// TwinCAT 3 PLC project Untitled1
// ProgramVersion: 3.1.4024.0
// libraries:
//   Tc2_MC2, * (Beckhoff Automation GmbH)
//   Tc2_Standard, * (Beckhoff Automation GmbH)
//   Tc2_System, * (Beckhoff Automation GmbH)
//   Tc3_Module, * (Beckhoff Automation GmbH)
//   VisuDialogs, * (System)
//   VisuSymbols,3.5.10.0,System
// project tree:
//   / GlobalTextList.TcGTLO, PlcTask.TcTTO (not stored), Visualization Manager.TcVMO (not stored)
//   GVLs/ BinSensorsFromPlc2.TcGVL, GVL.TcGVL (not stored), Inputs.TcGVL, MeasuringData.TcGVL, OpcuaData.TcGVL, Outputs.TcGVL, Steps.TcGVL
//   POUs/ AxisControl.TcPOU, BreedCalculation.TcPOU, Control24V.TcPOU, MAIN.TcPOU, PLC2Communicaton.TcPOU, SaveNewBinPosition.TcPOU, ServoManualMotion.TcPOU, SizeMeasure.TcPOU, TablePositions.TcPOU, WeightMeasure.TcPOU
//   VISUs/ HMI.TcVIS, InputsScreen.TcVIS, MainScreen.TcVIS, ManualMotionScreen.TcVIS, ServoMotionScreen.TcVIS
// real-time tasks:
//   TASK PlcTask: cycle T#10ms, priority 20, ADS port 350
// motion (NC):
//   TASK NC-Task 1 SAF: cycle T#2ms, priority 4, ADS port 501
//   TASK NC-Task 1 SVB: cycle T#10ms, priority 8, ADS port 511
//   AXIS Axis 1 (id 1)
//     Dynamic: Acceleration=120, Deceleration=120, Jerk=1000
//     Velo: SlowManual=20, FastManual=70, Maximum=150
//     OtherSettings: AllowMotionCmdToSlave=true
//     encoder EncType=1
//       EncPara: ScaleFactorNumerator=1
//         SoftEndMinControl: Enable=true, Range=-500
//         SoftEndMaxControl: Enable=true, Range=500
//     drive DrvType=5
//       Analog: VeloReferenz=100, TorqueSetpointScale=10, ScaleFactorActTorque=0.1
//       TimeComp: TaskDelayCycles=1
//     controller CtrType=1
//       CtrPara: PriorControlFactor=1
//         Observer: BandWidth=20
// variable links:
//   Untitled1/Untitled1 Instance <-> NC-Task 1 SAF/Axes/Axis 1
//     PlcTask Inputs/GVL.Axis.NcToPlc <-> Outputs/ToPlc
//     PlcTask Outputs/GVL.Axis.PlcToNc <-> Inputs/FromPlc

// ---- GVLs/BinSensorsFromPlc2.TcGVL
{attribute 'qualified_only'}
VAR_GLOBAL
	Bin1Full : BOOL := TRUE;
	Bin2Full : BOOL := TRUE;
	Bin3Full : BOOL := TRUE;
	Bin4Full : BOOL := TRUE;

END_VAR

// ---- GVLs/Inputs.TcGVL
{attribute 'qualified_only'}
VAR_GLOBAL
	Start_pos : BOOL;
	Size_measure_pos : BOOL;
	Weight_mes_pos : BOOL;
	Servo_table_pos : BOOL;
	Metal_sensor : BOOL;
	Grip_cyl_end_ext : BOOL;
	Grip_cyl_end_ret : BOOL;
	Cyl_at_table_ext : BOOL;
	Cyl_at_table_ret : BOOL;
	ES1 : BOOL;
	ES2 : BOOL;
	Size_measure : INT;
	Load_cell : INT;
	Grip_cyl_start_ext : BOOL;
	Grip_cyl_start_ret : BOOL;
	Control24VButton : BOOL;
	Metal_measure_pos : BOOL;
	End_pos_at_conveyor : BOOL;
	Item_left_the_table : BOOL;
END_VAR

// ---- GVLs/MeasuringData.TcGVL
{attribute 'qualified_only'}
VAR_GLOBAL
	AutomaticMode : BOOL;		
	StartConveyor : BOOL;	
	StopConveyor : BOOL;		
	ItemInTheSystem : BOOL; //If there is an item in the system
	ItemInTheSystemOnHmi : BOOL := TRUE; //If the variable true the text is invisible
	TableAtHome : BOOL;		
	TableAtBin1 : BOOL;		
	TableAtBin2 : BOOL;		
	TableAtBin3 : BOOL;		
	TableAtBin4 : BOOL;		
	ES1NC : BOOL := TRUE; //Emergency button for simulation
	ES2NC : BOOL := TRUE; //Emergency button for simulation
	ControlSupplyOK : BOOL; //Control 24V for simulation
	ControlSupplyOKOnHmi : BOOL := TRUE; //If the variable true the text is invisible
	SizeInCm : REAL;		
	MetalMaterial : BOOL;		
	WeightInKg : REAL;	
	Bin1Breed : BOOL; //Small and non metal
	Bin2Breed : BOOL; //Small and metal
	Bin3Breed : BOOL; //Large and not metal
	Bin4Breed : BOOL; //Large and metal
	Bin1BreedOnHmi : BOOL := TRUE; //If the variable true the text is invisible
	Bin2BreedOnHmi : BOOL := TRUE; //If the variable true the text is invisible
	Bin3BreedOnHmi : BOOL := TRUE; //If the variable true the text is invisible
	Bin4BreedOnHmi : BOOL := TRUE; //If the variable true the text is invisible
	HomePosition : LREAL;	
	Bin1Position : LREAL := 30.0;		
	Bin2Position : LREAL := 60.0;		
	Bin3Position : LREAL := 90.0;		
	Bin4Position : LREAL := 120.0;	
	MoveToBin1PositionByManual : BOOL;		
	MoveToBin2PositionByManual : BOOL;		
	MoveToBin3PositionByManual : BOOL;		
	MoveToBin4PositionByManual : BOOL;		
	MoveToHomeByManual : BOOL;		
	SaveNewPositionOfBin1 : BOOL;	
	SaveNewPositionOfBin2 : BOOL;		
	SaveNewPositionOfBin3 : BOOL;		
	SaveNewPositionOfBin4 : BOOL;		

END_VAR

// ---- GVLs/OpcuaData.TcGVL
{attribute 'qualified_only'}
VAR_GLOBAL
END_VAR

// ---- GVLs/Outputs.TcGVL
{attribute 'qualified_only'}
VAR_GLOBAL
	Green_light : BOOL;
	Yellow_light : BOOL;
	Red_light : BOOL;
	Move_grip_cyl_end_fwd : BOOL;
	Move_grip_cyl_end_bwd : BOOL;
	Move_cyl_at_table_fwd : BOOL;
	Move_cyl_at_table_bwd : BOOL;
	Conveyor_forward : BOOL;
	Conveyor_backward : BOOL;
	Move_grip_cyl_start_fwd : BOOL;
	Move_grip_cyl_start_bwd : BOOL;
	Blue_light : BOOL;

END_VAR

// ---- GVLs/Steps.TcGVL
{attribute 'qualified_only'}
VAR_GLOBAL
	ActualStep : BYTE := 1;
END_VAR

// ---- POUs/AxisControl.TcPOU
FUNCTION_BLOCK AxisControl
VAR_INPUT
	//Enable
	McPowerEnable : BOOL;
	//Jog
	JogForward : BOOL;
	JogBackward : BOOL;
	JogVelocity : LREAL;
	//Absolute move
	AbsolutePosition : LREAL;
	ExecuteMoveAbsoluteByManual : BOOL;
	ExecuteMoveAbsoluteByAutomatic : BOOL;
	MoveToBin1 : BOOL;
	MoveToBin2 : BOOL;
	MoveToBin3 : BOOL;
	MoveToBin4 : BOOL;
	//Home move
	ExecuteHomeByManual : BOOL;
	ExecuteHomeByAutomatic : BOOL;
END_VAR
VAR_OUTPUT
	//Position
	ActualPosition : LREAL;
	//Velocity
	ActualVelocity : LREAL;
END_VAR
VAR
	//Power
	McPower : MC_Power;
	McPowerError : BOOL;
	AxisStatus : BOOL;
	//JOG
	McJog : MC_Jog;

	//Relative
	McMoveRelative : MC_MoveRelative;
	ExecuteRelative : BOOL;
	RelativeDistance : LREAL;
	RelativeVelocity : LREAL;
	//Absolute
	McMoveAbsolute : MC_MoveAbsolute;
	ExecuteAbsolute : BOOL;
	AbsoluteVelocity : LREAL;
	//Velocity
	McMoveVelocity : MC_MoveVelocity;
	ExecuteVelocity : BOOL;
	Velocity : LREAL;
	//Home
	McHome: MC_Home;
	ExecuteHome : BOOL;
	HomeSensor : BOOL;
	//Stop
	McStop : MC_Stop;
	ExecuteStop : BOOL;
	//Halt
	McHalt: MC_Halt;
	ExecuteHalt : BOOL;
END_VAR

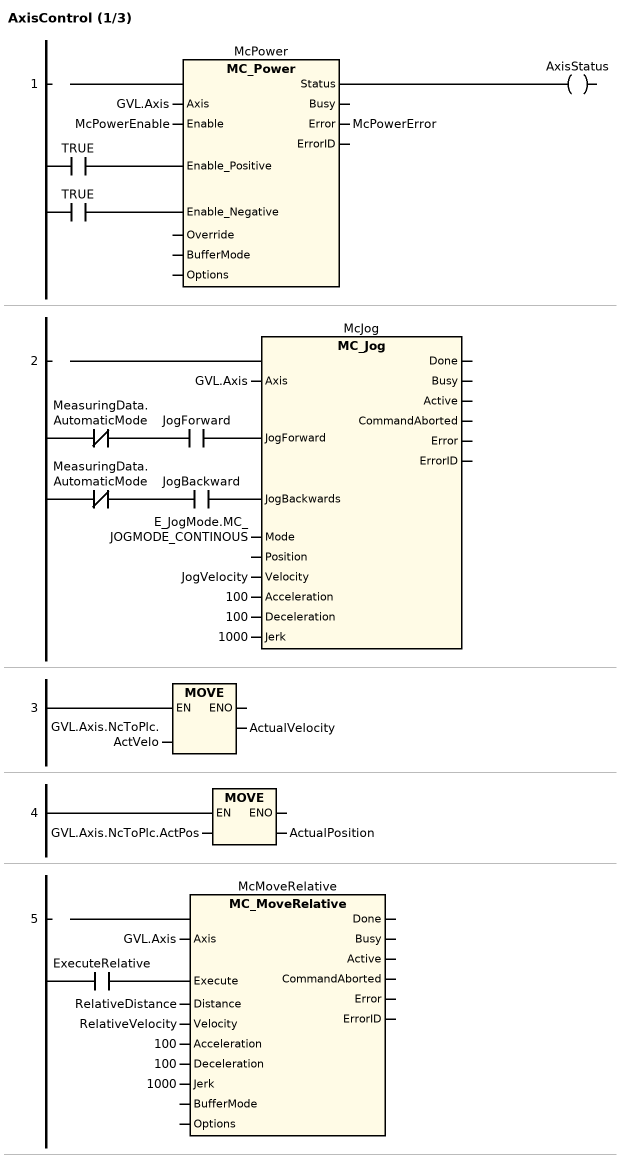
// NETWORK 1
McPower(
    Axis := GVL.Axis,
    Enable := McPowerEnable,
    Enable_Positive := TRUE,
    Enable_Negative := TRUE,
    Error => McPowerError); // MC_Power
AxisStatus := McPower.Status;

// NETWORK 2
McJog(
    Axis := GVL.Axis,
    JogForward := NOT MeasuringData.AutomaticMode AND JogForward,
    JogBackwards := NOT MeasuringData.AutomaticMode AND JogBackward,
    Mode := E_JogMode.MC_JOGMODE_CONTINOUS,
    Velocity := JogVelocity,
    Acceleration := 100,
    Deceleration := 100,
    Jerk := 1000); // MC_Jog

// NETWORK 3
ActualVelocity := GVL.Axis.NcToPlc.ActVelo;

// NETWORK 4
ActualPosition := GVL.Axis.NcToPlc.ActPos;

// NETWORK 5
McMoveRelative(
    Axis := GVL.Axis,
    Execute := ExecuteRelative,
    Distance := RelativeDistance,
    Velocity := RelativeVelocity,
    Acceleration := 100,
    Deceleration := 100,
    Jerk := 1000); // MC_MoveRelative

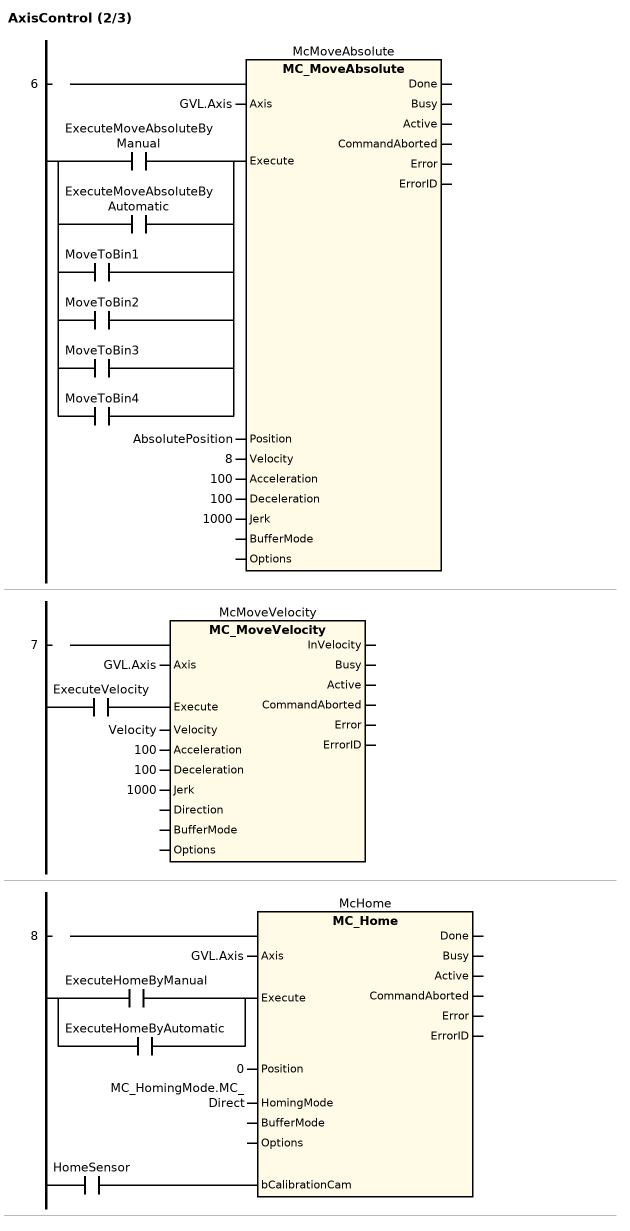
// NETWORK 6
McMoveAbsolute(
    Axis := GVL.Axis,
    Execute := ExecuteMoveAbsoluteByManual OR ExecuteMoveAbsoluteByAutomatic OR MoveToBin1 OR MoveToBin2 OR MoveToBin3 OR MoveToBin4,
    Position := AbsolutePosition,
    Velocity := 8,
    Acceleration := 100,
    Deceleration := 100,
    Jerk := 1000); // MC_MoveAbsolute

// NETWORK 7
McMoveVelocity(
    Axis := GVL.Axis,
    Execute := ExecuteVelocity,
    Velocity := Velocity,
    Acceleration := 100,
    Deceleration := 100,
    Jerk := 1000); // MC_MoveVelocity

// NETWORK 8
McHome(
    Axis := GVL.Axis,
    Execute := ExecuteHomeByManual OR ExecuteHomeByAutomatic,
    Position := 0,
    HomingMode := MC_HomingMode.MC_Direct,
    bCalibrationCam := HomeSensor); // MC_Home

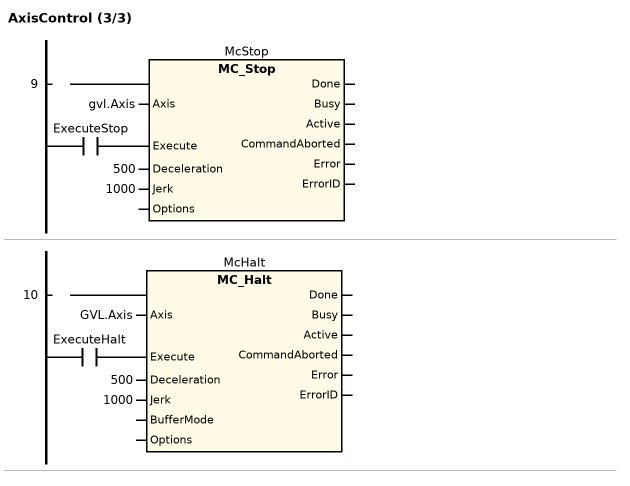
// NETWORK 9
McStop(Axis := gvl.Axis, Execute := ExecuteStop, Deceleration := 500, Jerk := 1000); // MC_Stop

// NETWORK 10
McHalt(Axis := GVL.Axis, Execute := ExecuteHalt, Deceleration := 500, Jerk := 1000); // MC_Halt

END_FUNCTION_BLOCK

// ---- POUs/BreedCalculation.TcPOU
FUNCTION BreedCalculation
VAR_INPUT
END_VAR
VAR

END_VAR


//Small and non metal. Bin1 breed
IF (MAIN.sizeMeasure.sizeInCm >= 10.0 AND MAIN.sizeMeasure.sizeInCm <= 20.0 AND MAIN.weightMeasure.weightInKg <= 5.0 AND
	NOT MeasuringData.MetalMaterial) THEN
	MeasuringData.Bin1Breed := TRUE;
	MeasuringData.Bin2Breed := FALSE;
	MeasuringData.Bin3Breed := FALSE;
	MeasuringData.Bin4Breed := FALSE;
	//Variables on the HMI
	MeasuringData.Bin1BreedOnHmi := FALSE;
	MeasuringData.Bin2BreedOnHmi := TRUE;
	MeasuringData.Bin3BreedOnHmi := TRUE;
	MeasuringData.Bin4BreedOnHmi := TRUE;
END_IF

//Small and metal. Bin2 breed
IF (MAIN.sizeMeasure.sizeInCm >= 10.0 AND MAIN.sizeMeasure.sizeInCm <= 20.0 AND MAIN.weightMeasure.weightInKg <= 5.0 AND
	MeasuringData.MetalMaterial) THEN
	MeasuringData.Bin1Breed := FALSE;
	MeasuringData.Bin2Breed := TRUE;
	MeasuringData.Bin3Breed := FALSE;
	MeasuringData.Bin4Breed := FALSE;
	//Variables on the HMI
	MeasuringData.Bin1BreedOnHmi := TRUE;
	MeasuringData.Bin2BreedOnHmi := FALSE;
	MeasuringData.Bin3BreedOnHmi := TRUE;
	MeasuringData.Bin4BreedOnHmi := TRUE;
END_IF

//Large and non metal. Bin3 breed
IF (MAIN.sizeMeasure.sizeInCm >= 20.0 AND MAIN.weightMeasure.weightInKg >= 5.1 AND
	NOT MeasuringData.MetalMaterial) THEN
	MeasuringData.Bin1Breed := FALSE;
	MeasuringData.Bin2Breed := FALSE;
	MeasuringData.Bin3Breed := TRUE;
	MeasuringData.Bin4Breed := FALSE;
	//Variables on the HMI
	MeasuringData.Bin1BreedOnHmi := TRUE;
	MeasuringData.Bin2BreedOnHmi := TRUE;
	MeasuringData.Bin3BreedOnHmi := FALSE;
	MeasuringData.Bin4BreedOnHmi := TRUE;
END_IF

//Large and metal. Bin4 breed
IF (MAIN.sizeMeasure.sizeInCm >= 20.0 AND MAIN.weightMeasure.weightInKg >= 5.1 AND
	MeasuringData.MetalMaterial) THEN
	MeasuringData.Bin1Breed := FALSE;
	MeasuringData.Bin2Breed := FALSE;
	MeasuringData.Bin3Breed := FALSE;
	MeasuringData.Bin4Breed := TRUE;
	//Variables on the HMI
	MeasuringData.Bin1BreedOnHmi := TRUE;
	MeasuringData.Bin2BreedOnHmi := TRUE;
	MeasuringData.Bin3BreedOnHmi := TRUE;
	MeasuringData.Bin4BreedOnHmi := FALSE;
END_IF

END_FUNCTION

// ---- POUs/MAIN.TcPOU
PROGRAM MAIN
VAR
	AxisControl : AxisControl;
	sizeMeasure : sizeMeasure;
	weightMeasure : WeightMeasure;
	control24V : Control24V;
	
	//Timers
	fbTon1 : TON;
	fbTon2 : TON;
	fbTon3 :TON;
	fbTon4 :TON;
	fbTon5 : TON;
	fbTon6 : TON;
	fbTon7 : TON;
	fbTp1 : TP;
	
	//Falling and rising edges
	startPosFallingEdge : F_TRIG;
	itemLeftTheTableFallingEdge : F_TRIG;
	
END_VAR

AxisControl();
sizeMeasure();
weightMeasure();

//Control 24V power supply
control24V();

//If there is 24V control supply, the servo is ready to operate
IF MeasuringData.ControlSupplyOK THEN
	AxisControl(McPowerEnable := TRUE);
ELSE
	AxisControl(McPowerEnable := FALSE);
END_IF

//Table positions
TablePositions();

//Save new bin position
SaveNewBinPosition();

//Breed calculation
BreedCalculation();

//Manual motion of servo
ServoManualMotion();

//PLC2 communication

//The blue light is on if there is 24V control supply.
IF MeasuringData.ControlSupplyOK THEN
	Outputs.Blue_light := TRUE;
ELSE
	Outputs.Blue_light := FALSE;
END_IF

//Start the system and the conveyor from HMI button.
//The yellow light is on.
IF MeasuringData.AutomaticMode AND MeasuringData.StartConveyor THEN
	fbTon1(IN := TRUE, PT := T#3S);
ELSE
	fbTon1(IN := FALSE);
END_IF

IF fbTon1.Q THEN
	Outputs.Yellow_light := TRUE;
	Outputs.Conveyor_forward := TRUE;
END_IF

//Halt the conveyor
IF MeasuringData.AutomaticMode AND MeasuringData.StopConveyor THEN
	Outputs.Conveyor_forward := FALSE;
END_IF

//Halt the servo motor

//Move gripping cylinder in start position backward.
//If there is no item in the system.
IF Steps.ActualStep = 1 AND Inputs.Start_pos THEN
	fbTon2(IN := TRUE, PT := T#3S);
ELSE
	fbTon2(IN := FALSE);
END_IF

IF fbTon2.Q AND NOT MeasuringData.ItemInTheSystem THEN
	Outputs.Move_grip_cyl_start_bwd := TRUE;
	Steps.ActualStep := 2;
END_IF

//After leaving the start position sensor, the system is in progress so there is an item in the system.
//The green light is on.
//The yellow light is off.
//Move gripping cylinder in start position forward.
startPosFallingEdge(CLK := Inputs.Start_pos);
IF startPosFallingEdge.Q THEN
	MeasuringData.ItemInTheSystem := TRUE;
	MeasuringData.ItemInTheSystemOnHmi := FALSE;
	Outputs.Green_light := TRUE;
	Outputs.Yellow_light := FALSE;
	Outputs.Move_grip_cyl_start_bwd := FALSE;
END_IF

//If the sensor active for two seconds, save the size in the data block.
IF Steps.ActualStep = 2 AND Inputs.Size_measure_pos THEN
	fbTon3(IN := TRUE, PT := T#3S);
ELSE
	fbTon3(IN := FALSE);
END_IF

IF fbTon3.Q THEN
	MeasuringData.SizeInCm := sizeMeasure.sizeInCm;
	Steps.ActualStep := 3;
END_IF

//Metal measure
IF Steps.ActualStep = 3 AND Inputs.Metal_measure_pos AND Inputs.Metal_sensor THEN
	MeasuringData.MetalMaterial := TRUE;
	Steps.ActualStep :=4 ;
END_IF

//Weight measure
IF Steps.ActualStep = 4 AND Inputs.Weight_mes_pos THEN
	fbTon4(IN := TRUE, PT := T#2S);
ELSE
	fbTon4(IN := FALSE);
END_IF

IF fbTon4.Q THEN
	MeasuringData.WeightInKg := weightMeasure.weightInKg;
	Steps.ActualStep := 5;
END_IF

//TCP/IP communication between the PLCs.
//If the end position sensor or sensor at the table are active, getting bin saturation data from PLC2.


//Retract gripping cylinder in end position
//If the sensor at conveyor is active for 1.5 seconds and the reed sensor is active and the certain bin is not full and the table is at home position.
//The state of bin sensors comes from PLC2.
IF Steps.ActualStep = 5 AND Inputs.End_pos_at_conveyor THEN
	fbTon5(IN := TRUE, PT := T#1.5S);
ELSE
	fbTon5(IN := FALSE);
END_IF

IF fbTon5.Q AND Inputs.Grip_cyl_end_ext AND MeasuringData.TableAtHome AND
	(
	(MeasuringData.Bin1Breed AND NOT BinSensorsFromPlc2.Bin1Full) OR
	(MeasuringData.Bin2Breed AND NOT BinSensorsFromPlc2.Bin2Full) OR
	(MeasuringData.Bin3Breed AND NOT BinSensorsFromPlc2.Bin3Full) OR
	(MeasuringData.Bin4Breed AND NOT BinSensorsFromPlc2.Bin4Full)
	)
	THEN
	
	Outputs.Move_grip_cyl_end_bwd := TRUE;
	Steps.ActualStep := 6;
END_IF

//Moving the servo controlled table to the appropriate position.
//If the item is already on the table, extending the cylinder in end position.
IF Inputs.Servo_table_pos THEN
	fbTon6(IN := TRUE, PT := T#2S);
ELSE
	fbTon6(IN := FALSE);
END_IF

IF fbTon6.Q THEN
	Outputs.Move_grip_cyl_end_bwd := FALSE;
END_IF

//Move to bin1
IF fbTon6.Q AND MeasuringData.Bin1Breed AND NOT BinSensorsFromPlc2.Bin1Full THEN
	AxisControl(AbsolutePosition := MeasuringData.Bin1Position);
	AxisControl(MoveToBin1 := TRUE);
ELSE
	AxisControl(AbsolutePosition := 0.0);
	AxisControl(MoveToBin1 := FALSE);
END_IF

//Move to bin2
IF fbTon6.Q AND MeasuringData.Bin2Breed AND NOT BinSensorsFromPlc2.Bin2Full THEN
	AxisControl(AbsolutePosition := MeasuringData.Bin2Position);
	AxisControl(MoveToBin2 := TRUE);
ELSE
	AxisControl(AbsolutePosition := 0.0);
	AxisControl(MoveToBin2 := FALSE);
END_IF

//Move to bin3
IF fbTon6.Q AND MeasuringData.Bin3Breed AND NOT BinSensorsFromPlc2.Bin3Full THEN
	AxisControl(AbsolutePosition := MeasuringData.Bin3Position);
	AxisControl(MoveToBin3 := TRUE);
ELSE
	AxisControl(AbsolutePosition := 0.0);
	AxisControl(MoveToBin3 := FALSE);
END_IF

//Move to bin4
IF fbTon6.Q AND MeasuringData.Bin4Breed AND NOT BinSensorsFromPlc2.Bin4Full THEN
	AxisControl(AbsolutePosition := MeasuringData.Bin4Position);
	AxisControl(MoveToBin4 := TRUE);
ELSE
	AxisControl(AbsolutePosition := 0.0);
	AxisControl(MoveToBin4 := FALSE);
END_IF

(*
Push the item into the proper bin then retract the cylinder.
Move the table back to home position.

There is no item in the system any more.
The next item can move forward from the beginning of the conveyor.
The green light goes off.
The yellow light goes on.
Reset the parameters of the item.
*)
IF Inputs.Servo_table_pos AND (
	(MeasuringData.Bin1Breed AND NOT BinSensorsFromPlc2.Bin1Full) OR
	(MeasuringData.Bin2Breed AND NOT BinSensorsFromPlc2.Bin2Full) OR
	(MeasuringData.Bin3Breed AND NOT BinSensorsFromPlc2.Bin3Full) OR
	(MeasuringData.Bin4Breed AND NOT BinSensorsFromPlc2.Bin4Full)
	)
	THEN
	
	fbTon7(IN := TRUE, PT := T#2S);
ELSE
	fbTon7(IN := FALSE);
END_IF

IF fbTon7.Q THEN
	Outputs.Move_cyl_at_table_fwd := TRUE;
END_IF

IF Inputs.Cyl_at_table_ext THEN
	Outputs.Move_cyl_at_table_fwd := FALSE;
END_IF

itemLeftTheTableFallingEdge(CLK := Inputs.Item_left_the_table);
IF itemLeftTheTableFallingEdge.Q THEN
	fbTp1(IN := TRUE, PT := T#1S);
ELSE
	fbTp1(IN := FALSE);
END_IF

IF fbTp1.Q THEN
	MeasuringData.ItemInTheSystem := FALSE;
	Outputs.Green_light := FALSE;
	Outputs.Yellow_light := TRUE;
	MeasuringData.SizeInCm := 0.0;
	MeasuringData.MetalMaterial := FALSE;
	MeasuringData.WeightInKg := 0.0;
	MeasuringData.ItemInTheSystemOnHmi := TRUE;
	MeasuringData.Bin1Breed := FALSE;
	MeasuringData.Bin1BreedOnHmi := TRUE;
	MeasuringData.Bin2Breed := FALSE;
	MeasuringData.Bin2BreedOnHmi := TRUE;
	MeasuringData.Bin3Breed := FALSE;
	MeasuringData.Bin3BreedOnHmi := TRUE;
	MeasuringData.Bin4Breed := FALSE;
	MeasuringData.Bin4BreedOnHmi := TRUE;
	
	IF NOT Inputs.Servo_table_pos AND Inputs.Cyl_at_table_ret THEN
		AxisControl(ExecuteHomeByAutomatic := TRUE);
	ELSE
		AxisControl(ExecuteHomeByAutomatic := FALSE);
	END_IF
ELSE
	AxisControl(ExecuteHomeByAutomatic := FALSE);
END_IF

END_PROGRAM

// ---- POUs/SizeMeasure.TcPOU
FUNCTION_BLOCK SizeMeasure
VAR_INPUT
END_VAR
VAR_OUTPUT
	//0-115cm
	sizeInCm : REAL;
END_VAR
VAR
	//0%-100%
	sizeInPercent : REAL;

    rawMin   : INT := 0;
    rawMax   : INT := 32767;
    scaledMin : REAL := 0.0;
    scaledMax : REAL := 115.0;
END_VAR

//Scaling
sizeInPercent := (scaledMax - scaledMin) / (rawMax - rawMin);
sizeInCm := scaledMin + (sizeInPercent * (inputs.Size_measure - rawMin));

END_FUNCTION_BLOCK

// ---- POUs/WeightMeasure.TcPOU
FUNCTION_BLOCK WeightMeasure
VAR_INPUT
END_VAR
VAR_OUTPUT
	//0-15kg
	weightInKg : REAL;
END_VAR
VAR
	//0%-100%
	weightInPercent : REAL;

    rawMin   : INT := 0;
    rawMax   : INT := 32767;
    scaledMin : REAL := 0.0;
    scaledMax : REAL := 15.0;
END_VAR

//Scaling
weightInPercent := (scaledMax - scaledMin) / (rawMax - rawMin);
weightInKg := scaledMin + (weightInPercent * (inputs.Load_cell - rawMin));

END_FUNCTION_BLOCK

// ---- POUs/Control24V.TcPOU
FUNCTION_BLOCK Control24V
VAR_INPUT
END_VAR
VAR_OUTPUT
END_VAR
VAR
	fbTon : TON;
END_VAR

//Control 24V for simulation
//This is the simulation of the safety circuit. Power supply for the output modules.
IF (MeasuringData.ES1NC AND MeasuringData.ES2NC AND Inputs.Control24VButton) THEN
	fbTon(IN := TRUE, PT := T#3S);
ELSE
	fbTon(IN := FALSE);
END_IF

MeasuringData.ControlSupplyOK := fbTon.Q;
MeasuringData.ControlSupplyOKOnHmi := NOT fbTon.Q;

END_FUNCTION_BLOCK

// ---- POUs/TablePositions.TcPOU
FUNCTION TablePositions
VAR_INPUT
END_VAR
VAR
END_VAR

//Home position
IF MAIN.AxisControl.ActualPosition = 0.0 THEN
	MeasuringData.TableAtHome := TRUE;
ELSIF MAIN.AxisControl.ActualPosition > 0.0 THEN
	MeasuringData.TableAtHome := FALSE;
END_IF

//Bin1 position
IF MAIN.AxisControl.ActualPosition >= 29.99 AND MAIN.AxisControl.ActualPosition <= 30.099 THEN
	MeasuringData.TableAtBin1 := TRUE;
ELSIF MAIN.AxisControl.ActualPosition < 29.99 OR MAIN.AxisControl.ActualPosition > 30.099 THEN
	MeasuringData.TableAtBin1 := FALSE;
END_IF

//Bin2 position
IF MAIN.AxisControl.ActualPosition >= 59.99 AND MAIN.AxisControl.ActualPosition <= 60.099 THEN
	MeasuringData.TableAtBin2 := TRUE;
ELSIF MAIN.AxisControl.ActualPosition < 59.99 OR MAIN.AxisControl.ActualPosition > 60.099 THEN
	MeasuringData.TableAtBin2 := FALSE;
END_IF

//Bin3 position
IF MAIN.AxisControl.ActualPosition >= 89.99 AND MAIN.AxisControl.ActualPosition <= 90.099 THEN
	MeasuringData.TableAtBin3 := TRUE;
ELSIF MAIN.AxisControl.ActualPosition < 89.99 OR MAIN.AxisControl.ActualPosition > 90.099 THEN
	MeasuringData.TableAtBin3 := FALSE;
END_IF

//Bin4 position
IF MAIN.AxisControl.ActualPosition >= 119.99 AND MAIN.AxisControl.ActualPosition <= 120.099 THEN
	MeasuringData.TableAtBin4 := TRUE;
ELSIF MAIN.AxisControl.ActualPosition < 119.99 OR MAIN.AxisControl.ActualPosition > 120.099 THEN
	MeasuringData.TableAtBin4 := FALSE;
END_IF

END_FUNCTION

// ---- POUs/SaveNewBinPosition.TcPOU
FUNCTION SaveNewBinPosition
VAR_INPUT
END_VAR
VAR
END_VAR

//New position of bin1
IF MeasuringData.SaveNewPositionOfBin1 THEN
	MeasuringData.Bin1Position := MAIN.AxisControl.ActualPosition;
END_IF
//New position of bin2
IF MeasuringData.SaveNewPositionOfBin2 THEN
	MeasuringData.Bin2Position := MAIN.AxisControl.ActualPosition;
END_IF
//New position of bin3
IF MeasuringData.SaveNewPositionOfBin3 THEN
	MeasuringData.Bin3Position := MAIN.AxisControl.ActualPosition;
END_IF
//New position of bin4
IF MeasuringData.SaveNewPositionOfBin4 THEN
	MeasuringData.Bin4Position := MAIN.AxisControl.ActualPosition;
END_IF

END_FUNCTION

// ---- POUs/ServoManualMotion.TcPOU
FUNCTION ServoManualMotion
VAR_INPUT
END_VAR
VAR
END_VAR

//Move to home
IF  NOT MeasuringData.AutomaticMode AND MeasuringData.MoveToHomeByManual THEN
	MAIN.AxisControl(ExecuteHomeByManual := TRUE);
ELSE
	MAIN.AxisControl(ExecuteHomeByManual := FALSE);
END_IF

//Move to bin1, bin2, bin3, bin4
IF NOT MeasuringData.AutomaticMode AND MeasuringData.MoveToBin1PositionByManual THEN
		MAIN.AxisControl(AbsolutePosition := MeasuringData.Bin1Position);
	ELSIF NOT MeasuringData.AutomaticMode AND MeasuringData.MoveToBin2PositionByManual THEN
		MAIN.AxisControl(AbsolutePosition := MeasuringData.Bin2Position);
	ELSIF NOT MeasuringData.AutomaticMode AND MeasuringData.MoveToBin3PositionByManual THEN
		MAIN.AxisControl(AbsolutePosition := MeasuringData.Bin3Position);
	ELSIF NOT MeasuringData.AutomaticMode AND MeasuringData.MoveToBin4PositionByManual THEN
		MAIN.AxisControl(AbsolutePosition := MeasuringData.Bin4Position);
	ELSE
		MAIN.AxisControl(AbsolutePosition := 0.0);
END_IF


//If one of the button is clicked on the HMI
IF (NOT MeasuringData.AutomaticMode AND MeasuringData.MoveToBin1PositionByManual) OR
	(NOT MeasuringData.AutomaticMode AND MeasuringData.MoveToBin2PositionByManual) OR
	(NOT MeasuringData.AutomaticMode AND MeasuringData.MoveToBin3PositionByManual) OR
	(NOT MeasuringData.AutomaticMode AND MeasuringData.MoveToBin4PositionByManual) THEN
	MAIN.AxisControl(ExecuteMoveAbsoluteByManual := TRUE);
ELSE
	MAIN.AxisControl(ExecuteMoveAbsoluteByManual := FALSE);
END_IF

END_FUNCTION

// ---- POUs/PLC2Communicaton.TcPOU
FUNCTION_BLOCK PLC2Communicaton
VAR_INPUT
END_VAR
VAR_OUTPUT
END_VAR
VAR
END_VAR

END_FUNCTION_BLOCK

// ---- GlobalTextList.TcGTLO
TEXTLIST GlobalTextList
  489 = '%.0f'
  236 = '%.2f'
  710 = '%0.f'
  10 = '24V OK'
  115 = 'Actual position'
  154 = 'Automatic/Manual'
  868 = 'Bin1'
  891 = 'Bin2'
  170 = 'Bin3'
  250 = 'Bin4'
  150 = 'Breed'
  192 = 'Breed1'
  405 = 'Breed2'
  103 = 'Data'
  689 = 'Drive Control'
  693 = 'Drive enable'
  124 = 'Enter velocity'
  777 = 'Halt motion'
  543 = 'Home'
  965 = 'Home+'
  423 = 'Inputs'
  670 = 'Item in the'
  434 = 'Item in the '
  309 = 'Item in the system'
  235 = 'Jog velocity'
  326 = 'Jog+'
  694 = 'Jog-'
  924 = 'Jog-+'
  401 = 'Label'
  392 = 'Lights'
  95 = 'Manual control'
  679 = 'Manual motion'
  507 = 'Measuring system'
  503 = 'Metal'
  174 = 'Move absolute'
  964 = 'Move home'
  708 = 'Move relative'
  588 = 'Move velocity'
  925 = 'Position'
  468 = 'Power'
  863 = 'Reset'
  541 = 'Save new position'
  449 = 'Servo'
  776 = 'Servo motion'
  644 = 'Size'
  429 = 'Sorting system'
  231 = 'Start conveyor'
  351 = 'Stop conveyor'
  536 = 'Stop motion'
  27 = 'Type absolute pos'
  85 = 'Type absolute velocity'
  97 = 'Type relative pos'
  81 = 'Type relative velocity'
  642 = 'Type velocity'
  655 = 'Velocity'
  341 = 'Vlamai'
  218 = 'Weight'
END_TEXTLIST

// ---- VISUs/HMI.TcVIS
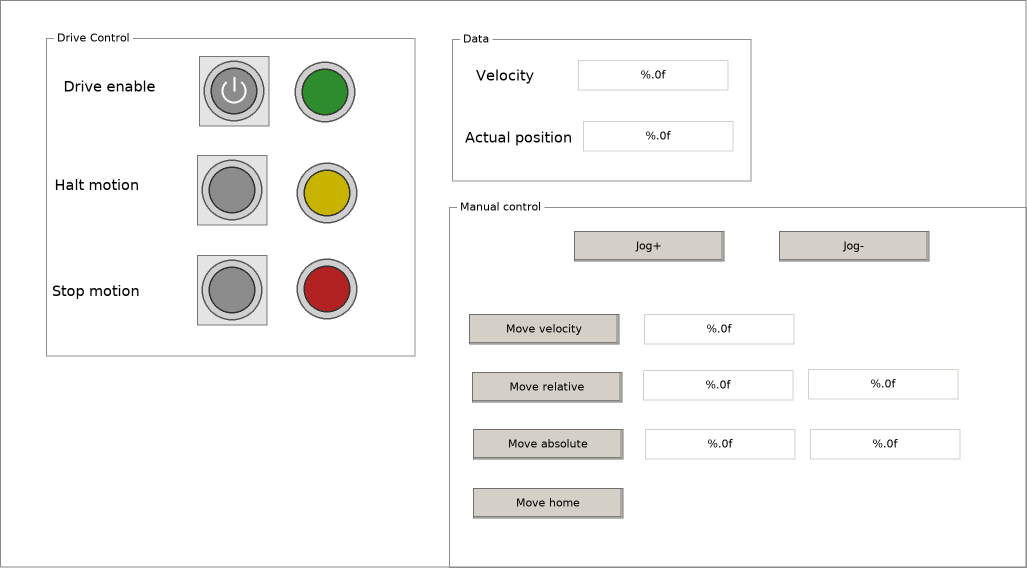
VISUALIZATION HMI  // 1027x568
    GroupBox (46,30 369x326), "Drive Control"
        PowerSwitch (153,26 70x70), variable: MAIN.AxisControl.McPowerEnable, behaviour: TOGGLE, style: Switch-PowerSwitch-Gray
        Lamp1 (244,27 70x70), variable: MAIN.AxisControl.AxisStatus, style: Lamp-Lamp1-Green
        PushSwitch (151,125 70x70), variable: MAIN.AxisControl.ExecuteHalt, behaviour: TOGGLE, style: Switch-PushSwitch-Gray
        PushSwitch (151,225 70x70), variable: MAIN.AxisControl.ExecuteStop, behaviour: TOGGLE, style: Switch-PushSwitch-Gray
        Lamp1 (246,128 70x70), variable: MAIN.AxisControl.McHalt.Done, style: Lamp-Lamp1-Yellow
        Lamp1 (246,224 70x70), variable: MAIN.AxisControl.McStop.Done, style: Lamp-Lamp1-Red
    Label (22,170 150x30), "Halt motion"
    Label (21,276 150x30), "Stop motion"
    Label (44,66 131x41), "Drive enable"
    GroupBox (452,31 299x150), "Data"
        Label (6,32 94x25), "Velocity"
        Textfield (126,29 150x30), "%.0f", text variable: MAIN.AxisControl.ActualVelocity
        Label (11,95 111x23), "Actual position"
        Textfield (131,90 150x30), "%.0f", text variable: MAIN.AxisControl.ActualPosition
    GroupBox (449,199 578x369), "Manual control"
        Button (125,32 150x30), "Jog+"
            OnMouseDown: toggle MAIN.AxisControl.JogForward
        Button (330,32 150x30), "Jog-"
            OnMouseDown: toggle MAIN.AxisControl.JogBackward
        Button (20,115 150x30), "Move velocity"
            OnMouseDown: toggle MAIN.AxisControl.ExecuteVelocity
        Textfield (195,115 150x30), "%.0f", tooltip "Type velocity", text variable: MAIN.AxisControl.Velocity
            OnMouseClick: write the text variable via Edit, min 0, max 50
        Button (23,173 150x30), "Move relative"
            OnMouseDown: toggle MAIN.AxisControl.ExecuteRelative
        Textfield (194,171 150x30), "%.0f", tooltip "Type relative pos", text variable: MAIN.AxisControl.RelativeDistance
            OnMouseClick: write the text variable via Edit
        Button (24,230 150x30), "Move absolute"
            OnMouseDown: toggle MAIN.AxisControl.ExecuteAbsolute
        Textfield (196,230 150x30), "%.0f", tooltip "Type absolute pos", text variable: MAIN.AxisControl.AbsolutePosition
            OnMouseClick: write the text variable via Edit
        Button (24,289 150x30), "Move home"
            OnMouseDown: toggle MAIN.AxisControl.ExecuteHome
        Textfield (359,170 150x30), "%.0f", tooltip "Type relative velocity", text variable: MAIN.AxisControl.RelativeVelocity
            OnMouseClick: write the text variable via Edit
        Textfield (361,230 150x30), "%.0f", tooltip "Type absolute velocity", text variable: MAIN.AxisControl.AbsoluteVelocity
            OnMouseClick: write the text variable via Edit
END_VISUALIZATION

// ---- VISUs/InputsScreen.TcVIS
VISUALIZATION InputsScreen  // 2x2
END_VISUALIZATION

// ---- VISUs/MainScreen.TcVIS
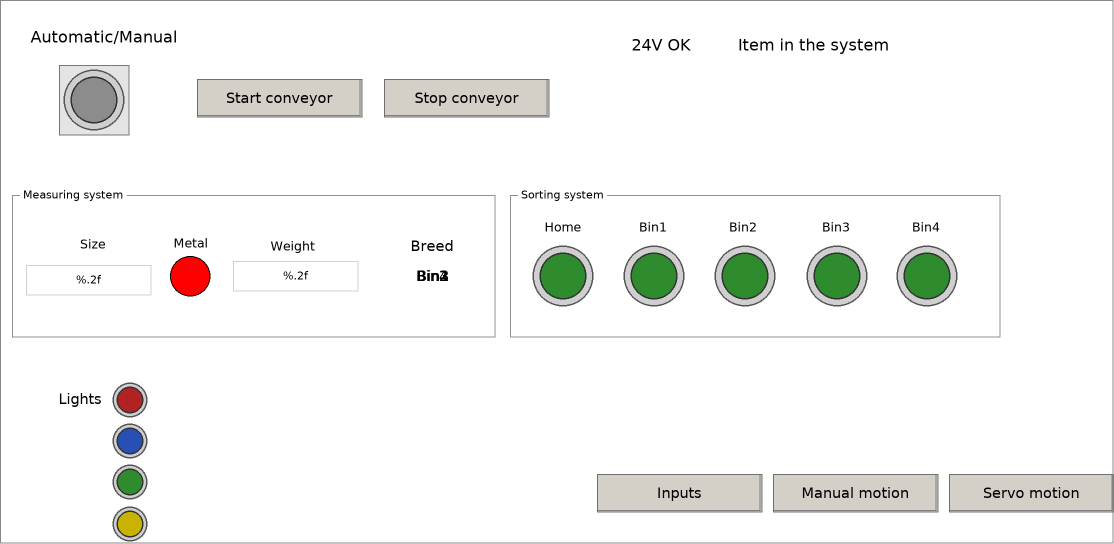
VISUALIZATION MainScreen  // 1114x544
    PushSwitch (59,65 70x70), variable: MeasuringData.AutomaticMode, behaviour: TOGGLE, style: Switch-PushSwitch-Gray
    Label (13,18 182x38), "Automatic/Manual"
    Button (197,79 165x38), "Start conveyor"
        OnMouseDown: execute { MeasuringData.StartConveyor := TRUE; }
        OnMouseUp: execute { MeasuringData.StartConveyor := FALSE; }
    Button (384,79 165x38), "Stop conveyor"
        OnMouseDown: execute { MeasuringData.StopConveyor := TRUE; }
        OnMouseUp: execute { MeasuringData.StopConveyor := FALSE; }
    Label (595,26 132x38), "24V OK", invisible if: MeasuringData.ControlSupplyOKOnHmi
    Label (729,26 169x38), "Item in the system", invisible if: MeasuringData.ItemInTheSystemOnHmi
    GroupBox (12,187 483x150), "Measuring system"
        Textfield (14,78 125x30), "%.2f", text variable: MeasuringData.SizeInCm
        Label (6,42 150x30), "Size"
        Ellipse (158,69 40x40), colour toggle: MeasuringData.MetalMaterial
        Label (138,41 82x30), "Metal"
        Textfield (221,74 125x30), "%.2f", text variable: MeasuringData.WeightInKg
        Label (240,44 82x30), "Weight"
        Label (379,44 82x30), "Breed"
        Label (380,74 82x30), "Bin1", invisible if: MeasuringData.Bin1BreedOnHmi
        Label (380,74 82x30), "Bin3", invisible if: MeasuringData.Bin3BreedOnHmi
        Label (379,74 82x30), "Bin4", invisible if: MeasuringData.Bin4BreedOnHmi
    GroupBox (510,187 490x150), "Sorting system"
        Lamp1 (18,54 70x70), variable: MeasuringData.TableAtHome, style: Lamp-Lamp1-Green
        Lamp1 (109,54 70x70), variable: MeasuringData.TableAtBin1, style: Lamp-Lamp1-Green
        Lamp1 (200,54 70x70), variable: MeasuringData.TableAtBin2, style: Lamp-Lamp1-Green
        Lamp1 (292,54 70x70), variable: MeasuringData.TableAtBin3, style: Lamp-Lamp1-Green
        Lamp1 (382,54 70x70), variable: MeasuringData.TableAtBin4, style: Lamp-Lamp1-Green
        Label (12,25 82x30), "Home"
        Label (102,25 82x30), "Bin1"
        Label (192,25 82x30), "Bin2"
        Label (285,25 82x30), "Bin3"
        Label (375,25 82x30), "Bin4"
    Button (597,474 165x38), "Inputs"
    Button (773,474 165x38), "Manual motion"
    Button (949,474 165x38), "Servo motion"
    Label (39,384 82x30), "Lights"
    Lamp1 (110,380 40x40), variable: Outputs.Red_light, style: Lamp-Lamp1-Red
    Lamp1 (110,421 40x40), variable: Outputs.Blue_light, style: Lamp-Lamp1-Blue
    Lamp1 (110,462 40x40), variable: Outputs.Green_light, style: Lamp-Lamp1-Green
    Lamp1 (110,504 40x40), variable: Outputs.Yellow_light, style: Lamp-Lamp1-Yellow
    Label (391,261 82x30), "Bin2", invisible if: MeasuringData.Bin2BreedOnHmi
END_VISUALIZATION

// ---- VISUs/ManualMotionScreen.TcVIS
VISUALIZATION ManualMotionScreen  // 2x2
END_VISUALIZATION

// ---- VISUs/ServoMotionScreen.TcVIS
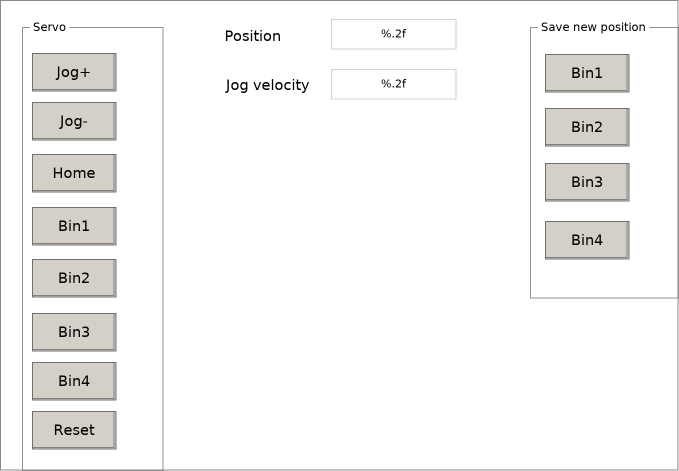
VISUALIZATION ServoMotionScreen  // 679x471
    GroupBox (22,19 141x452), "Servo"
        Button (10,34 84x38), "Jog+"
            OnMouseDown: execute { MAIN.AxisControl.JogForward := TRUE; }
            OnMouseUp: execute { MAIN.AxisControl.JogForward := FALSE; }
        Button (10,83 84x38), "Jog-"
            OnMouseDown: execute { MAIN.AxisControl.JogBackward := TRUE; }
            OnMouseUp: execute { MAIN.AxisControl.JogBackward := FALSE; }
        Button (10,135 84x38), "Home"
            OnMouseDown: execute { MAIN.AxisControl.ExecuteHomeByManual := TRUE; }
            OnMouseUp: execute { MAIN.AxisControl.ExecuteHomeByManual := FALSE; }
        Button (10,188 84x38), "Bin1"
            OnMouseDown: execute { MeasuringData.MoveToBin1PositionByManual := TRUE; }
            OnMouseUp: execute { MeasuringData.MoveToBin1PositionByManual := FALSE; }
        Button (10,240 84x38), "Bin2"
            OnMouseDown: execute { MeasuringData.MoveToBin2PositionByManual := TRUE; }
            OnMouseUp: execute { MeasuringData.MoveToBin2PositionByManual := FALSE; }
        Button (10,294 84x38), "Bin3"
            OnMouseDown: execute { MeasuringData.MoveToBin3PositionByManual := TRUE; }
            OnMouseUp: execute { MeasuringData.MoveToBin3PositionByManual := FALSE; }
        Button (10,343 84x38), "Bin4"
            OnMouseDown: execute { MeasuringData.MoveToBin4PositionByManual := TRUE; }
            OnMouseUp: execute { MeasuringData.MoveToBin4PositionByManual := FALSE; }
        Button (10,392 84x38), "Reset"
    Label (212,21 82x30), "Position"
    Label (212,70 112x30), "Jog velocity"
    Textfield (331,19 125x30), "%.2f", text variable: MAIN.AxisControl.ActualPosition
    Textfield (331,69 125x30), "%.2f", text variable: MAIN.AxisControl.JogVelocity
    GroupBox (530,19 149x279), "Save new position"
        Button (15,35 84x38), "Bin1"
            OnMouseDown: execute { MeasuringData.SaveNewPositionOfBin1 := TRUE; }
            OnMouseUp: execute { MeasuringData.SaveNewPositionOfBin1 := FALSE; }
        Button (15,89 84x38), "Bin2"
            OnMouseDown: execute { MeasuringData.SaveNewPositionOfBin2 := TRUE; }
            OnMouseUp: execute { MeasuringData.SaveNewPositionOfBin2 := FALSE; }
        Button (15,144 84x38), "Bin3"
            OnMouseDown: execute { MeasuringData.SaveNewPositionOfBin3 := TRUE; }
            OnMouseUp: execute { MeasuringData.SaveNewPositionOfBin3 := FALSE; }
        Button (15,202 84x38), "Bin4"
            OnMouseDown: execute { MeasuringData.SaveNewPositionOfBin4 := TRUE; }
            OnMouseUp: execute { MeasuringData.SaveNewPositionOfBin4 := FALSE; }
END_VISUALIZATION
